PROGRAM Signals
VAR
	fbTimer1: TON;
	TON_0: TON;
END_VAR

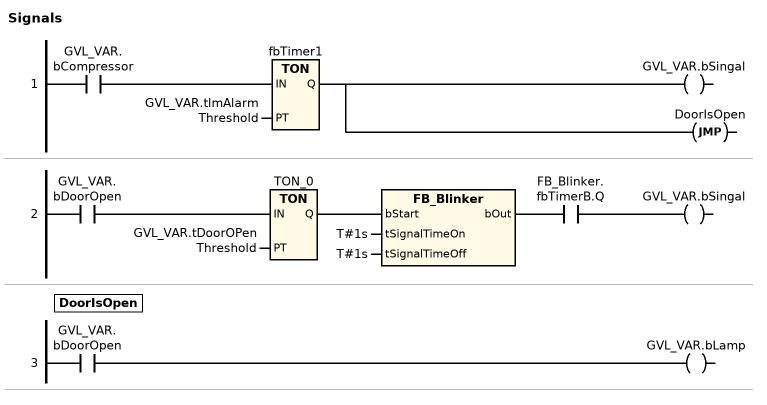
// NETWORK 1
fbTimer1(IN := GVL_VAR.bCompressor, PT := GVL_VAR.tlmAlarmThreshold); // TON
GVL_VAR.bSingal := fbTimer1.Q;
IF fbTimer1.Q THEN JMP DoorIsOpen; END_IF

// NETWORK 2
TON_0(IN := GVL_VAR.bDoorOpen, PT := GVL_VAR.tDoorOPenThreshold); // TON
FB_Blinker(bStart := TON_0.Q, tSignalTimeOn := T#1s, tSignalTimeOff := T#1s);
GVL_VAR.bSingal := FB_Blinker.bOut AND FB_Blinker.fbTimerB.Q;

// NETWORK 3
DoorIsOpen:
GVL_VAR.bLamp := GVL_VAR.bDoorOpen;

END_PROGRAM

(* stored: Version 1.1.0.1, ProductVersion 3.1.4024.12
   POU Signals: Id {dd828172-10b3-494e-afda-ba8efbe9b66c}, SpecialFunc None *)
